# EPICS autosave request: newstep/NSC200_settings.req
$(P)$(M):COMDISABLE
$(P)$(M):TWSIZE
